DATA_BLOCK "TON"
VAR
  TON : Array[0..100] of TON_TIME;
  CTU : Array[0..20] of IEC_DCOUNTER;
  P : Array[0..20] of Bool;
END_VAR
BEGIN
END_DATA_BLOCK
